TYPE ST_PTM :
STRUCT
(* General PTM Structure
Each PTM might have a serial control structure, but all will have a general supervisory control structure

NOTE: This is an archetype, use an extension of this structure for a specific pump (or make one).

*)

(* Controls *)
	i_xRunSW : BOOL;
	q_RunDO : BOOL;

(* Readbacks *)
	xExtRunOk	:	BOOL; (* also a control *)
	i_xAccel	:	BOOL;
	i_xAtSpd	:	BOOL;
	i_iCurSpd	:	DINT;
	
	xCommTimeout	:	BOOL := TRUE;  (* Initialized true since we haven't talked to pump yet *)
(* Alarm Outputs *)
	xFault		:	BOOL; //Note, for Ebara this is *false* in a fault condition!
	xWarn		:	BOOL; (* warning *)
	
(* IWS instructions *)
	xActive	:	BOOL; // this bit is set to add the pump to the system
	iPumpGrp 	:	INT; // all members of a pump group start at the same time

END_STRUCT
END_TYPE

(* stored: Version 1.1.0.1, ProductVersion 3.1.4018.5
   DUT ST_PTM: Id {800c0744-7104-483e-92b7-6bb5c958de58} *)
